Universal Robots PolyScope program: Socket_control.urp

Program Socket_control (installation=default directory=/programs/usbdisk createdIn=3.1.17195.0 lastSavedIn=3.10.0.76181 robotSerialNumber=2019330557)
Calibrated DH parameters: a=[0.000115, -0.205025, -0.212758, -0.000082, 0.00002, 0]; d=[0.151838, 61.855759, -55.531221, -6.212403, 0.085388, 0.082596]; alpha=[1.571271, -0.002138, 0.002223, 1.571866, -1.571624, 0]; deltaTheta=[0.000009, -0.572803, 0.638806, -0.065963, 0.000015, 0.000024]
BeforeStart
  IP := "192.168.1.111"
  PORT := 888
  open := socket_open(IP,PORT)
  Loop While (checkContinuously=false) expression=open≟ False
    open := socket_open(IP,PORT)
  Script: pos = get_actual_tcp_pose()
  Script: jpos = get_actual_joint_positions()
  Script: msg = "stop"
  Script: cmdMsg = "stop"
  Script: dynamic =  True
  Script: msgFloat = [0,0.0,0.0,0.0,0.0,0.0,0.0]
  Script: list_rq = [0,0,0,0]
  URCap Gripper Activate (Robotiq_Grippers, Robotiq Inc.) dataModel(ResetAndActivateKey=false)
Robot Program (runOnlyOnce=false)
  Script file /programs/socketControl_v2.script
    | while True:
    | 
    | 	if (dynamic == True):
    | 		if (cmdMsg == "stop"):
    | 			end_freedrive_mode()
    | 			stopj(2)
    | 		elif (cmdMsg == "recordj"):
    | 			freedrive_mode()
    | 
    | 		elif (cmdMsg == "pservoj"):
    | 			pos = p[msgFloat[1],msgFloat[2],msgFloat[3],msgFloat[4],msgFloat[5],msgFloat[6]]
    | 			jpos = get_inverse_kin(pos)
    | 			servoj(jpos)
    | 
    | 		elif (cmdMsg == "pservoc"):
    | 			pos = p[msgFloat[1],msgFloat[2],msgFloat[3],msgFloat[4],msgFloat[5],msgFloat[6]]
    | 			servoc(pos)
    | 
    | 		elif (cmdMsg == "jservoj"):
    | 			jpos = [msgFloat[1],msgFloat[2],msgFloat[3],msgFloat[4],msgFloat[5],msgFloat[6]]
    | 			servoj(jpos)
    | 		end
    | 	end
    | 
    | 	if (dynamic == False):
    | 		if (cmdMsg == "jmovej"):
    | 			jpos = [msgFloat[1],msgFloat[2],msgFloat[3],msgFloat[4],msgFloat[5],msgFloat[6]]
    | 			movej(jpos)
    | 			socket_send_string("UR:done")
    | 		elif (cmdMsg == "pmovep"):
    | 			pos = p[msgFloat[1],msgFloat[2],msgFloat[3],msgFloat[4],msgFloat[5],msgFloat[6]]
    | 			movep(pos)
    | 			socket_send_string("UR:done")
    | 		elif (cmdMsg == "pmovej"):
    | 			pos = p[msgFloat[1],msgFloat[2],msgFloat[3],msgFloat[4],msgFloat[5],msgFloat[6]]
    | 			jpos = get_inverse_kin(pos)
    | 			movej(jpos)
    | 			socket_send_string("UR:done")
    | 		elif (cmdMsg == "Rmovej"):
    | 			nowPosj = get_target_joint_positions()
    | 			jpos = [nowPosj[0]+msgFloat[1],nowPosj[1]+msgFloat[2],nowPosj[2]+msgFloat[3],nowPosj[3]+msgFloat[4],nowPosj[4]+msgFloat[5],nowPosj[5]+msgFloat[6]]
    | 			movej(jpos)
    | 			socket_send_string("UR:done")
    | 		elif (cmdMsg == "Rmovep"):
    | 			nowPos = get_actual_tcp_pose()
    | 			pos = p[nowPos[0]+msgFloat[1],nowPos[1]+msgFloat[2],nowPos[2]+msgFloat[3],nowPos[3]+msgFloat[4],nowPos[4]+msgFloat[5],nowPos[5]+msgFloat[6]]
    | 			movep(pos)
    | 			socket_send_string("UR:done")
    | 		elif (cmdMsg == "gripper"):
    | 			list_rq[0] = msgFloat[1]*1000
    | 			list_rq[1] = msgFloat[2]*1000
    | 			list_rq[2] = msgFloat[3]*1000
    | 			rq_set_force(list_rq[1])
    | 			rq_set_speed(list_rq[2])
    | 			rq_move(list_rq[0])
    | 			while(rq_is_motion_complete() == False):
    | 			end
    | 			socket_send_string("UR:done")
    | 		elif (cmdMsg == "recordj"):
    | 			freedrive_mode()
    | 		end
    | 		dynamic = True
    | 	end
    | end
Thread Thread_1 (runOnlyOnce=false trackProgramExecution=false)
  Script file /programs/sub_socket_read.script
    | #//thread will stuck and wait cmd
    | while True:
    |     msg = socket_read_string() #//stuck
    | 
    |     if msg == "stop":
    |         cmdMsg = "stop"
    |         dynamic = True
    |         socket_send_string(get_actual_tcp_pose())
    |     elif msg == "recordj":
    |         cmdMsg = "recordj"
    |         dynamic = True
    |         socket_send_string(get_actual_joint_positions())
    |     elif msg == "pservoj":
    |         dynamic = True
    |         socket_send_string("UR:"+ cmdMsg)
    |         msgFloat = socket_read_ascii_float(6)
    |         while msgFloat[0] != 6:
    |             msgFloat = socket_read_ascii_float(6)
    |         end
    |         socket_send_string(get_actual_tcp_pose())
    |         cmdMsg = "pservoj"
    |     elif msg == "pservoc":
    |         cmdMsg = "pservoc"
    |         dynamic = True
    |         socket_send_string("UR:"+ cmdMsg)
    |         msgFloat = socket_read_ascii_float(6)
    |         while msgFloat[0] != 6:
    |             msgFloat = socket_read_ascii_float(6)
    |         end
    |         socket_send_string(get_actual_tcp_pose())
    |     elif msg == "jservoj":
    |         dynamic = True
    |         socket_send_string("UR:"+ cmdMsg)
    |         msgFloat = socket_read_ascii_float(6)
    |         while msgFloat[0] != 6:
    |             msgFloat = socket_read_ascii_float(6)
    |         end
    |         socket_send_string(get_actual_joint_positions())
    |         cmdMsg = "jservoj"
    | 	elif msg == "jmovej":
    |         cmdMsg = "jmovej"
    |         socket_send_string("UR:"+ cmdMsg)
    |         msgFloat = socket_read_ascii_float(6)
    |         while msgFloat[0] != 6:
    |             msgFloat = socket_read_ascii_float(6)
    |         end
    | 		dynamic = False
    | 	elif msg == "pmovep":
    |         cmdMsg = "pmovep"
    |         socket_send_string("UR:"+ cmdMsg)
    |         msgFloat = socket_read_ascii_float(6)
    |         while msgFloat[0] != 6:
    |             msgFloat = socket_read_ascii_float(6)
    |         end
    |         dynamic = False
    |     elif msg == "pmovej":
    |         cmdMsg = "pmovej"
    |         socket_send_string("UR:"+ cmdMsg)
    |         msgFloat = socket_read_ascii_float(6)
    |         while msgFloat[0] != 6:
    |             msgFloat = socket_read_ascii_float(6)
    |         end
    | 		dynamic = False
    |     elif msg == "Rmovej":
    |         cmdMsg = "Rmovej"
    |         socket_send_string("UR:"+ cmdMsg)
    |         msgFloat = socket_read_ascii_float(6)
    |         while msgFloat[0] != 6:
    |             msgFloat = socket_read_ascii_float(6)
    |         end
    | 		dynamic = False
    | 	elif msg == "Rmovep":
    |         cmdMsg = "Rmovep"
    |         socket_send_string("UR:"+ cmdMsg)
    |         msgFloat = socket_read_ascii_float(6)
    |         while msgFloat[0] != 6:
    |             msgFloat = socket_read_ascii_float(6)
    |         end
    | 		dynamic = False
    | 	elif msg == "gripper":
    |         cmdMsg = "gripper"
    |         socket_send_string("UR:"+ cmdMsg)
    |         msgFloat = socket_read_ascii_float(6)
    |         while msgFloat[0] != 6:
    |             msgFloat = socket_read_ascii_float(6)
    |         end
    |         dynamic = False
    | 	end
    | end
